Staubli VAL3: cycleStatus.dtx

public ActionItem aActionTime
  [0]
    num nDistance = 1
    num nMoveId = 3
    num nTimeId
    num nPointId
    InstrItem iInstr[3]
      [0]
        string sType
        string sData
      [1]
        string sType
        string sData
      [2]
        string sType
        string sData
    string sIdTraj = "POINT place"
public InstrItem iToSuperV
  [0]
    string sType = "PROG"
    string sData = "home"
InstrItem tcpInstr[3]
  [0]
    string sType = "OUT"
    string sData = "bOut0>ON"
  [1]
    string sType = "OUT"
    string sData = "bOut1>OFF"
  [2]
    string sType
    string sData
Trajectory tTrajCycle
  [0]
    TrajectoryItem tSuper[3]
      [0]
        num distance
        num moveType = 1
        num nTime
        num nStop
        num nTcpAction
        string comment = "appro"
        bool toStop
        mdesc nom_speed = {tmax=1000, rmax=9999, leave=30, reach=30}
        InstrItem iInstr[3]
          [0]
            string sType
            string sData
          [1]
            string sType
            string sData
          [2]
            string sType
            string sData
        num nMoveId
      [1]
        num distance
        num moveType = 1
        num nTime
        num nStop
        num nTcpAction = 1
        string comment = "point"
        bool toStop = true
        mdesc nom_speed = {tmax=1000, rmax=9999, leave=30, reach=30}
        InstrItem iInstr[3]
          [0]
            string sType
            string sData
          [1]
            string sType
            string sData
          [2]
            string sType
            string sData
        num nMoveId
      [2]
        num distance
        num moveType = 1
        num nTime
        num nStop
        num nTcpAction
        string comment = "depart"
        bool toStop
        mdesc nom_speed = {tmax=1000, rmax=9999, leave=30, reach=30}
        InstrItem iInstr[3]
          [0]
            string sType
            string sData
          [1]
            string sType
            string sData
          [2]
            string sType
            string sData
        num nMoveId = 127
    string sID = "POINT pick"
    num nId
bool bActionMutex
public bool bAutoON
public bool bCALL
public bool bCycle
public bool bEnding
public bool bGOTO
public bool bHomeLoaded = true
public bool bHoming
public bool bIsHome
bool bLogMutex
public bool bMotionToken
public bool bMoveStopped
public bool bMutex
public bool bPause
public bool bPausePLC
public bool bShowMessage
public bool bSimulation
public bool bStop
public bool bToEnd
public bool bToHome
public bool bToPause
public bool bToStart
public bool bToStop
public bool bTrackEnable
public bool bTraj = true
public bool bWait
public bool bWritingToLog
public num nClockAction = 7230.098
public num nCycleTime = 1.833
public num nEmergency
public num nEvent
public num nIdPercentage = 5.617
public num nInterfaceToSV = -1
public num nLastIdPoint
public num nLastTimer = 5.715
public num nPoint = 2
public num nProcessType = 1
public num nProg
public num nTime = 7764.435
public num nToSuperV = -1
num nTollerance = 150
public num nWorkingMode = 4
public num nWorkingStatus = 2
pointRx pTollerance = {x=387.992409, y=64.919473, z=-164.968083, rx=0.107448, ry=178.01498, rz=42.225142, shoulder=lefty, elbow=epositive, wrist=wpositive, fatherId=world[0]}
public progItem pCycleProg
  [0]
    InstrItem iEvent[2]
      [0]
        string sType = "POINT"
        string sData = "pick"
      [1]
        string sType = "POINT"
        string sData = "place"
    string sID = "pick_place"
public string sLastAction = "OUT bOut0>OFF"
public string sToShow
public string sTraj
public string sTrajItem
ActionItem aActionTCP
  [0]
    num nDistance
    num nMoveId
    num nTimeId
    num nPointId
    InstrItem iInstr[3]
      [0]
        string sType
        string sData
      [1]
        string sType
        string sData
      [2]
        string sType
        string sData
    string sIdTraj
ActionItem aActionPoint
  [0]
    num nDistance
    num nMoveId
    num nTimeId
    num nPointId
    InstrItem iInstr[3]
      [0]
        string sType
        string sData
      [1]
        string sType
        string sData
      [2]
        string sType
        string sData
    string sIdTraj
public bool bActionRunning
ActionItem aAction
  [0]
    num nDistance
    num nMoveId
    num nTimeId
    num nPointId
    InstrItem iInstr[3]
      [0]
        string sType
        string sData
      [1]
        string sType
        string sData
      [2]
        string sType
        string sData
    string sIdTraj
public string sLog
public num nTimeMould[2]
